{attribute 'linkalways'} 
{attribute 'no_explicit_call' := 'This FB is a CLASS and must be accessed using methods or properties'}
{attribute 'enable_dynamic_creation'}
FUNCTION_BLOCK _USINT EXTENDS NumericDatatypeBase
VAR
	localData : USINT;
	activeData : REFERENCE TO USINT REF= localData;
END_VAR

PROPERTY PUBLIC Address : PVOID
GET
Address := ADR(activeData);
END_GET
END_PROPERTY

METHOD PUBLIC ClearReference
VAR_INPUT
END_VAR
activeData REF= localData;
END_METHOD

METHOD PUBLIC Clone : I_Datatype
VAR
    pClone : POINTER TO _USINT;
END_VAR
pClone := __NEW(_USINT(InitialValue := Value));
Clone := pClone^;
END_METHOD

METHOD FB_init : BOOL
VAR_INPUT
	bInitRetains : BOOL; // if TRUE, the retain variables are initialized (warm start / cold start)
	bInCopyCode : BOOL;  // if TRUE, the instance afterwards gets moved into the copy code (online change)
	InitialValue : USINT;
END_VAR
localData := InitialValue;
END_METHOD

PROPERTY PUBLIC IsFloat : BOOL
GET
IsFloat := FALSE;
END_GET
END_PROPERTY

PROPERTY PUBLIC IsSigned : BOOL
GET
IsSigned := FALSE;
END_GET
END_PROPERTY

METHOD PUBLIC MakeReferenceTo
VAR_INPUT
	ReferenceTarget : REFERENCE TO USINT;
END_VAR
activeData REF= ReferenceTarget;
END_METHOD

PROPERTY PUBLIC MaxValue : USINT
GET
MaxValue :=  DatatypeLimits.USINT_MAX_VALUE;
END_GET
END_PROPERTY

PROPERTY PUBLIC MinValue : USINT
GET
MinValue := DatatypeLimits.USINT_MIN_VALUE;
END_GET
END_PROPERTY

METHOD PROTECTED SerializeMaxValue
VAR_INPUT
	Serializer : I_Serializer;
END_VAR
Serializer.AddUsint(MaxValue);
END_METHOD

METHOD PROTECTED SerializeMinValue
VAR_INPUT
	Serializer : I_Serializer;
END_VAR
Serializer.AddUsint(MinValue);
END_METHOD

METHOD PUBLIC SerializeWith
VAR_INPUT
	Serializer : I_Serializer;
END_VAR
Serializer.AddUsint(activeData);
END_METHOD

PROPERTY PUBLIC Size : UDINT
GET
Size := SIZEOF(activeData);
END_GET
END_PROPERTY

METHOD TryDeserializeFrom : BOOL
VAR_INPUT
	Deserializer : I_Deserializer;
	Feedback : I_DeserializerFeedback;
END_VAR
TryDeserializeFrom := Deserializer.TryGetUsint(activeData, Feedback);
END_METHOD

METHOD TryMakeReferenceTo : BOOL
VAR_INPUT
	Target : I_Datatype;
END_VAR
VAR
	pTargetData : POINTER TO USINT;
END_VAR
IF NOT (Target.TypeName = TypeName) THEN
	RETURN;
END_IF

pTargetData := Target.Address;
activeData REF= pTargetData^;
TryMakeReferenceTo := TRUE;
END_METHOD

PROPERTY PUBLIC TypeName : T_MAXSTRING
GET
TypeName := 'USINT';
END_GET
END_PROPERTY

PROPERTY PUBLIC Value : USINT
GET
Value := activeData;
END_GET
SET
activeData := Value;
END_SET
END_PROPERTY

END_FUNCTION_BLOCK

(* stored: Version 1.1.0.1, ProductVersion 3.1.4024.12
   POU _USINT: Id {2936c95f-0287-41d7-b6a8-2b7cc2f494b2}, SpecialFunc None
   Folder Constructor: Id {b1e072c1-e060-495b-b682-613a6948e498}
   Folder Protected: Id {63834cec-4b59-4bf7-b146-fd1db6627c09}
   Property Address: Id {eece26d4-7e24-4c9c-add3-bfe3505c449a}
   Get Get: Id {c86e5216-aa63-414b-baa4-d83a2e3fa3de}
   Method ClearReference: Id {d0a32cfd-eab8-43fb-aeea-80cd30155e3d}
   Method Clone: Id {c466b556-d782-497e-ae59-243a4d0fd9f7}
   Method FB_init: Id {6404e0a6-5a2e-4c13-9e28-5fc2c03dd1a7}
   Property IsFloat: Id {2844c20e-2660-4869-b5ee-c56423b82cf8}
   Get Get: Id {57c687bc-4571-46c4-b92b-89c9624a2986}
   Property IsSigned: Id {663be363-2359-45c4-95c8-d9bc359daa27}
   Get Get: Id {a780054b-fe40-4050-99a3-0b45bab541c5}
   Method MakeReferenceTo: Id {cded812a-ecd5-4a6d-b9ff-e1b1daa6cd56}
   Property MaxValue: Id {6f5d2c26-3837-4f01-ac00-5a3508b05aac}
   Get Get: Id {dee68e37-23aa-425d-9583-4b4ad957f153}
   Property MinValue: Id {d820967c-3263-4f3d-bdcf-d4b8f9cf406c}
   Get Get: Id {d31879ab-b824-4f28-8414-f9335df3fffd}
   Method SerializeMaxValue: Id {9725683f-ae03-47ec-bfac-ec86e4c675e3}
   Method SerializeMinValue: Id {7d154fe6-1aef-445c-8c05-fa24a7bc4578}
   Method SerializeWith: Id {d9a763a5-08f5-4fcb-b142-0e514cf8ac5b}
   Property Size: Id {42ae505a-6f95-4e28-9e21-a8ccbc25bb5e}
   Get Get: Id {9f509d37-2e98-4722-9398-7cbd6377cbac}
   Method TryDeserializeFrom: Id {87acf17c-5bb2-4fb8-ab02-65fd76bbc9dd}
   Method TryMakeReferenceTo: Id {c7abae44-d2e6-4339-be01-bfcd075c87d7}
   Property TypeName: Id {ac00c49e-a50d-4410-b871-652bc7d060cb}
   Get Get: Id {9848f3a9-5483-43b1-a13d-6aa2728312a4}
   Property Value: Id {2d122a0f-2b21-4399-baea-07c867bb9c85}
   Get Get: Id {b666fb7f-38f2-4e55-a6f8-fba8b183369a}
   Set Set: Id {0dba600b-f09f-4ca6-be7a-5363e6f54089} *)
